FUNCTION_BLOCK Stopping EXTENDS Vanguard_WaferDetection.State
VAR
	ShutdownState : INT;
	ChannelControl : I_VisionChannelControl;
END_VAR

METHOD Executing : BOOL
CASE ShutdownState OF		
	0: //unkown conditions
		IF ChannelControl.StopVision() THEN
			ShutdownState := 1;
		END_IF
	1:
		Executing := TRUE;
		ShutdownState := 0;
END_CASE
END_METHOD

METHOD SetDependencies : BOOL
VAR_INPUT
	Control : I_VisionChannelControl;
END_VAR
ChannelControl := Control;
END_METHOD

END_FUNCTION_BLOCK

(* stored: Version 1.1.0.1
   POU Stopping: Id {4fde9158-fba4-42ed-b5ed-64b93305fb65}, SpecialFunc None
   Method Executing: Id {4be63fc8-f26d-4763-b7b8-780de5f6f461}
   Method SetDependencies: Id {2ba7f496-ec23-4aee-8f61-426e3400d8f0} *)
